FUNCTION_BLOCK FbFilterNaN //Фильтр NaN и Inf для чисел REAL.

//      DbFilterNaN
//    +-------------+
//    | FbFilterNaN |
// ->-|In        Out|->-
//    |        Alarm|-
//    +-------------+

VAR_INPUT //Входные переменные, сохраняемые.
In:REAL := 0.0; //Вход.
END_VAR

VAR_OUTPUT //Выходные переменные, сохраняемые.
Out   :REAL := 0.0  ; //Выход.
Alarm :BOOL := FALSE; //Флаг ошибки.
END_VAR

//Если In==(NaN или Inf или -Inf) то Out=0 иначе Out=In.
//DW#16#7F800000=DW#2#01111111_10000000_00000000_00000000
//Стандарт IEEE 754.
IF ((REAL_TO_DWORD(In) AND DW#16#7F800000) = DW#16#7F800000) THEN
Out   := 0.0;
Alarm := TRUE;
ELSE
Out   := In;
Alarm := FALSE;
END_IF;

END_FUNCTION_BLOCK

//  +---------+
//  | GNU GPL |
//  +---------+
//  |
//  |
//  .= .-_-. =.
// ((_/)o o(\_))
//  `-'(. .)`-'
//  |/| \_/ |\
//  ( |     | )
//  /"\_____/"\
//  \__)   (__/
// @COPYLEFT ALL WRONGS RESERVED :)
// Author: VA
// Contacts: DIY.PLC.314@gmail.com
// License: GNU GPL v2
